VAR_GLOBAL CONSTANT
	MAX_DIMENSIONS : INT := 3; (*Valid values are 1, 2, 3*)
END_VAR

(* stored: Version 1.1.0.1, ProductVersion 3.1.0.36
   GVL PLC_Interpolation_Parameters: Id {e191df13-0972-4bb0-9175-ad1b9d379ce0}, ParameterList True *)
